// TIA Portal V20 export
FUNCTION_BLOCK "FB_Recipe"   // FB81, SCL
{ S7_Optimized_Access := 'TRUE' }
// stored: AutoNumber false, MemoryReserve 100, SetENOAutomatically false
BEGIN
   REGION Description header 
       //==================================================================================
       // POSALUX Swiss SA / (C) Copyright 2026
       //----------------------------------------------------------------------------------
       // Title: FB_Recipe
       // Comment/Function: 
       //
       // Author: Fabien WALDT
       // Engineering: TIA Portal v20
       //----------------------------------------------------------------------------------
       // Change log table:
       // Version  | Date     | Expert in charge | Changes applied
       // ---------|----------|------------------|------------------------------------
       // 00.00.01 | 20260427 | WFA              | First released version
       // ==================================================================================
   END_REGION

   REGION Current
       "DB_OPC_Recipe".Current.RecipeId := "DB_OPC_Recipe".Current.RecipeId;
       "DB_OPC_Recipe".Current.RecipeVersionGuid := "DB_OPC_Recipe".Current.RecipeVersionGuid;
   END_REGION

   REGION Data
       "DB_OPC_Recipe".Data.LaserJobListName := "DB_OPC_Recipe".Data.LaserJobListName;
       "DB_OPC_Recipe".Data.RecipeId := "DB_OPC_Recipe".Data.RecipeId;
       "DB_OPC_Recipe".Data.RecipeName := "DB_OPC_Recipe".Data.RecipeName;
       "DB_OPC_Recipe".Data.RecipeVersionGuid := "DB_OPC_Recipe".Data.RecipeVersionGuid;

       // Station 1
       // General \ Detections \ WorkPart
       "DB_OPC_Recipe".Data.Station1.General.Detections.WorkPart.Max := "DB_OPC_Recipe".Data.Station1.General.Detections.WorkPart.Max;
       "DB_OPC_Recipe".Data.Station1.General.Detections.WorkPart.Min := "DB_OPC_Recipe".Data.Station1.General.Detections.WorkPart.Min;
       // General \ GasPressure
        "DB_OPC_Recipe".Data.Station1.General.GazPressure.WorkLaserDefault := "DB_OPC_Recipe".Data.Station1.General.GazPressure.WorkLaserDefault;
   END_REGION

   REGION TransfertToPlc
       IF "DB_OPC_Recipe".TransferToPlc THEN
           "DB_OPC_Recipe".Current.RecipeId := "DB_OPC_Recipe".Data.RecipeId;
           "DB_OPC_Recipe".Current.RecipeVersionGuid := "DB_OPC_Recipe".Data.RecipeVersionGuid;
           "DB_Scanner".sScannerComm.iJobListName := "DB_OPC_Recipe".Data.LaserJobListName;
       //    "DB_HMISetting".GasAssistSetPoint := LREAL_TO_REAL("DB_OPC_Recipe".Data.Station1.General.GazPressure.WorkLaserDefault);   WAF A LIBERER QUAND RECETTE OK
       //    "DB_GestionFixture".sFixturePartControl.iProdOK_LimHigh := LREAL_TO_REAL("DB_OPC_Recipe".Data.Station1.General.Detections.WorkPart.Max);  WAF A LIBERER QUAND RECETTE OK
       //    "DB_GestionFixture".sFixturePartControl.iProdOK_LimLow := LREAL_TO_REAL("DB_OPC_Recipe".Data.Station1.General.Detections.WorkPart.Min);   WAF A LIBERER QUAND RECETTE OK
           "DB_OPC_Recipe".TransferToPlc := FALSE;
       END_IF;
   END_REGION
END_FUNCTION_BLOCK
